FUNCTION Convert_UDINT_TO_STRING : BOOL
VAR_INPUT
	in : UDINT;
	out : REFERENCE TO STRING;
END_VAR
VAR
	converted : STRING;
END_VAR

converted := UDINT_TO_STRING(in);

IF (STRING_TO_UDINT(converted) <> in) THEN
	RETURN;
END_IF

out := converted;
Convert_UDINT_TO_STRING := TRUE;

END_FUNCTION

(* stored: Version 1.1.0.1, ProductVersion 3.1.4024.12
   POU Convert_UDINT_TO_STRING: Id {d1cc6183-f6ad-4e95-840a-ae7792613b35}, SpecialFunc None *)
